{attribute 'qualified_only'}
{attribute 'strict'}
TYPE E_Airpad :
(
	eDepressurize := 0,
    eAirpadOnMoveRequest := 1,
    eAirpadOnError := 2
);
END_TYPE

(* stored: Version 1.1.0.1
   EnumerationTextList E_Airpad: Id {46d4770e-f67e-0cc8-2f93-73eb81df36b2} *)
